// TIA Portal V19 export
FUNCTION "WR_Done" : Date_And_Time   // FC171, LAD
// stored: SetENOAutomatically false
   VAR_INPUT
      done : Bool;
   END_VAR
   VAR CONSTANT
      empty : Date_And_Time;
   END_VAR
BEGIN

REGION Network 1 (SCL)
   IF #done THEN 
       #"WR_Done" := "Now"();
   ELSE
       #"WR_Done" := #empty;
   END_IF;
   ENO := TRUE;
END_REGION
END_FUNCTION
